Universal Robots PolyScope program: LE02 SocketComms.urp

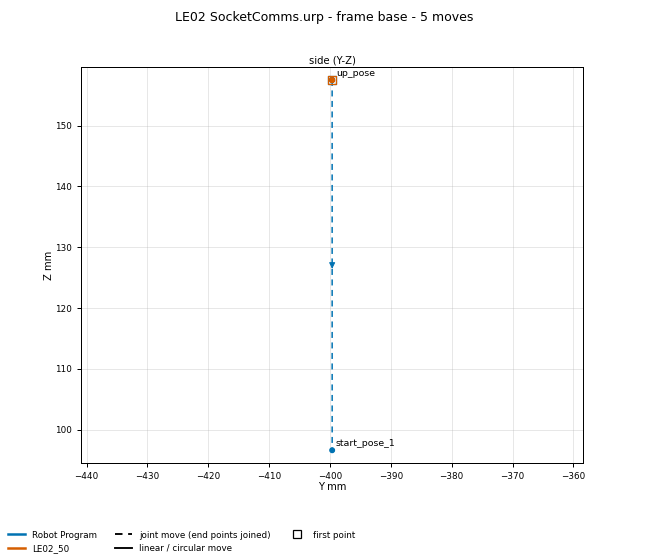
[picture p0: tool path of LE02 SocketComms.urp in frame base, 5 of 6 moves have a stored position in this frame; points joined in program order, loops and branches not executed]
Program LE02 SocketComms (installation=default directory=/programs/LE createdIn=5.7.0.90932 lastSavedIn=5.9.1.1031110 robotSerialNumber=20195501059)
Calibrated DH parameters: a=[0.000146, -0.418764, -0.053981, 0.000058, -0.000023, 0]; d=[0.162545, 37.319448, -206.067439, 168.881546, 0.09955, 0.099464]; alpha=[1.57004, -0.001979, 0.002304, 1.570607, -1.57066, 0]; deltaTheta=[0, -0.174616, -1.258233, 1.432844, -0.000001, 0]
BeforeStart
  URCap Gripper Activate (Robotiq_Grippers, Robotiq Inc.) dataModel(ResetAndActivateKey=false)
  start_pose := get_actual_tcp_pose()
  MoveJ speed 60 deg/s, acceleration 80 deg/s^2 (useActiveTCP=true) feature=Base
    Waypoint Waypoint (Variable): variable=start_pose
  Script: socket_close()
  Wait Sleep waitTime=0.25
  socket_is_open := False
  command_index := 0
Robot Program (runOnlyOnce=false)
  command_index := command_index+1
  Loop While (checkContinuously=false) expression=socket_is_open ≟  False
    socket_is_open := socket_open("192.168.0.252", 30000)
    Wait Sleep waitTime=0.5
  command := socket_read_ascii_float(5)
  response := "Unknown command"
  If command[0]≟5
    Script: socket_send_line("robot_running=True")
    Switch expression=command[1]
      Case (caseValue=1)
        MoveL speed 250 mm/s, acceleration 1200 mm/s^2 (useActiveTCP=true) feature=Base
          Waypoint up_pose: TCP in base x=296.6 y=-399.647 z=157.491 mm, rx=0.0004 ry=0.0085 rz=-0.0046 rad; joints [111.254, -87.197, 110.424, -113.021, 269.593, 201.526] deg; TCP offset x=0 y=0 z=175 mm, rx=3.1416 ry=0 rz=0 rad
        response := "moved up"
      Case (caseValue=2)
        MoveJ speed 60 deg/s, acceleration 80 deg/s^2 (useActiveTCP=true) feature=Base
          Waypoint start_pose_1: TCP in base x=296.589 y=-399.642 z=96.63 mm, rx=0.0004 ry=0.0085 rz=-0.0046 rad; joints [111.249, -83.001, 115.86, -122.649, 269.604, 201.537] deg
        response := "moved down"
      Case (caseValue=3)
        URCap Gripper (Robotiq_Grippers, Robotiq Inc.) dataModel(position=100.0, force=100.0, speed=100.0, positionInDouble=100.0, forceInDouble=100.0, speedInDouble=100.0, slaveIds=[9], blocking=true)
        response := "close"
      Case (caseValue=4)
        URCap Gripper (Robotiq_Grippers, Robotiq Inc.) dataModel(position=0.0, force=100.0, speed=100.0, positionInDouble=0.0, forceInDouble=100.0, speedInDouble=100.0, slaveIds=[9], blocking=true)
        response := "open"
      Case (caseValue=50)
        Call LE02_50
      Case (caseValue=98)
        response := "socket reset"
      Case (caseValue=99)
        response := "exiting"
      Case (caseValue=2147483647)
        response := "unknown command"
    Script: socket_send_line("robot_response=" + response + "#robot_running=False")
    If command[1]≟98
      Wait Sleep waitTime=0.5
      Script: socket_close()
      socket_is_open := False
    If command[1]≟99
      Wait Sleep waitTime=0.5
      Script: socket_close()
      socket_is_open := False
      Halt
  Else 
    command_index := command_index+1
    Script: socket_set_var("robot_index", command_index)
SubProgram -> LE02_50
SubProgram LE02_50 (keepSynchronizedWithDisk=true) programFile=/programs/LE/LE02_50.urp
  'Rev 2021_12_02am 01'
  MoveL speed 250 mm/s, acceleration 1200 mm/s^2 (useActiveTCP=true) feature=Base
    Waypoint Vertical_1: TCP in base x=296.586 y=-399.638 z=157.461 mm, rx=0.0001 ry=0 rz=-0.0068 rad; joints [110.998, -87.379, 110.673, -113.28, 270.04, 201.399] deg
    Waypoint Tilted_2: TCP in base x=296.604 y=-399.668 z=157.504 mm, rx=-0.5593 ry=0.007 rz=-0.0068 rad; joints [119.721, -93.557, 131.941, -156.668, 254.371, 206.211] deg
    Set DigitalOutput pin=digital_out[2]; digitalValue=1
    Wait Sleep waitTime=1
    Set DigitalOutput pin=digital_out[2]; digitalValue=0
    Waypoint Vertical_2: TCP in base x=296.586 y=-399.638 z=157.461 mm, rx=0.0001 ry=0 rz=-0.0068 rad; joints [110.998, -87.379, 110.673, -113.28, 270.04, 201.399] deg
    response := "50 success"
